// TIA Portal V16 export
// export: Created 2022-04-06T03:32:48.1224576Z, ExportSetting WithDefaults, DisplayName Totally Integrated Automation Portal, DisplayVersion V16 Update 4, DisplayName TIA Portal Version Control Interface, DisplayVersion V16 Update 2, DisplayName TIA Portal Openness, DisplayVersion V16 Update 4, DisplayName SINAMICS Startdrive Advanced, DisplayVersion V16, DisplayName SINAMICS Startdrive G130, G150, S120, S150, SINAMICS MV, S210, DisplayVersion V16, DisplayName SINAMICS Startdrive G110M, G120, G120C, G120D, G120P, DisplayVersion V16, DisplayName STEP 7 Professional, DisplayVersion V16 Update 4, DisplayName STEP 7 Safety, DisplayVersion V16, DisplayName WinCC Professional, DisplayVersion V16 Update 4
FUNCTION_BLOCK "fbRoomHVAC"   // FB7, LAD
{ S7_Optimized_Access := 'TRUE' }
VERSION : 0.1
// stored: AutoNumber true, IsIECCheckEnabled false, IsRetainMemResEnabled false, MemoryReserve 100, SetENOAutomatically false, UDAEnableTagReadback false
   VAR
      Temperature_Cooling { ExternalVisible := 'False'} : "fbAlarmedSetpoint";
      Humidity { ExternalVisible := 'False'} : "fbAlarmedSetpoint";
      CO2 { S7_SetPoint := 'True'} : "fbAlarmedSetpoint";
   END_VAR
   VAR RETAIN
      Controls { ExternalVisible := 'False'} : Struct
         rHeatingSP { ExternalVisible := 'False'} : Real := 55.0;
         bResetAlarm { ExternalVisible := 'False'} : Bool;
         bResetModbus { ExternalVisible := 'False'} : Bool;
      END_STRUCT;
      Status { ExternalVisible := 'False'; ExternalWritable := 'False'} : Struct
         bModbusError { ExternalVisible := 'False'; ExternalWritable := 'False'} : Bool;
         wLastModbusErrorCode { ExternalVisible := 'False'; ExternalWritable := 'False'} : Word;
      END_STRUCT;
      Config { ExternalVisible := 'False'} : Struct
         ModbusServerAddr { ExternalVisible := 'False'} : IP_V4;   // IP address for Modbus TCP server
         ID { ExternalVisible := 'False'} : UInt := 81;   // Unique ID for connection, also used as port number on PLC
      END_STRUCT;
   END_VAR
   VAR
      TCPConnection { ExternalAccessible := 'False'; ExternalVisible := 'False'; ExternalWritable := 'False'} : TCON_IP_v4;
      fbModbusTCPClient_Instance { ExternalAccessible := 'False'; ExternalVisible := 'False'; ExternalWritable := 'False'} : "fbModbusTCPClient";
      Read_Discrete { ExternalAccessible := 'False'; ExternalVisible := 'False'; ExternalWritable := 'False'} : Array[0..0] of "udtModbusValBool";
      Write_Discrete { ExternalAccessible := 'False'; ExternalVisible := 'False'; ExternalWritable := 'False'} : Array[0..0] of "udtModbusValBool";
      Read_Registers { ExternalAccessible := 'False'; ExternalVisible := 'False'; ExternalWritable := 'False'} : Array[0..2] of "udtModbusValReal";
      Write_Registers { ExternalAccessible := 'False'; ExternalVisible := 'False'; ExternalWritable := 'False'} : Array[0..2] of "udtModbusValReal";
      TON_ModbusReset { S7_SetPoint := 'True'} : TON_TIME;
      mbreset { ExternalAccessible := 'False'; ExternalVisible := 'False'; ExternalWritable := 'False'} : Bool;
      TP_ModbusResetPulse { S7_SetPoint := 'True'} : TP_TIME;
   END_VAR
   VAR CONSTANT
      cFakeScaling : Int := 150;
      cRoomTempIndex : Int := 0;
      cHumidityIndex : Int := 1;
      cCO2Index : Int := 2;
   END_VAR
   // Temperature_Cooling.arrSetpoints[1].rSetpoint := 75.0;
   // Humidity.arrSetpoints[1].rSetpoint := 55.0;
   // Config.ModbusServerAddr.ADDR[1] := 10;
   // Config.ModbusServerAddr.ADDR[2] := 1;
   // Config.ModbusServerAddr.ADDR[3] := 0;
   // Config.ModbusServerAddr.ADDR[4] := 8;
   // TCPConnection.ConnectionType := 11;
   // TCPConnection.ActiveEstablished := true;
   // TCPConnection.RemoteAddress.ADDR[1] := 10;
   // TCPConnection.RemoteAddress.ADDR[2] := 1;
   // TCPConnection.RemoteAddress.ADDR[3] := 2;
   // TCPConnection.RemoteAddress.ADDR[4] := 8;
   // TCPConnection.RemotePort := 502;
   // TCPConnection.LocalPort := 1001;
BEGIN

REGION Network 1 (SCL): Set connection parameters
   #TCPConnection.InterfaceId := "Local~PROFINET_interface_1"; // PLC ethernet port
   #TCPConnection.ID := UINT_TO_WORD(#Config.ID);
   #TCPConnection.ConnectionType := 11; // TCP
   #TCPConnection.ActiveEstablished := TRUE;
   #TCPConnection.RemoteAddress := #Config.ModbusServerAddr;
   #TCPConnection.RemotePort := 502; // Default for Modbus TCP
   #TCPConnection.LocalPort := #Config.ID;
END_REGION

REGION Network 2 (SCL): Reset Modbus on Error

   #mbreset := #TON_ModbusReset.Q;
   #TON_ModbusReset(IN := #Status.bModbusError AND NOT #mbreset,
                    PT := T#10S);

   #TP_ModbusResetPulse(IN:=#mbreset,
                        PT:=T#5S,
                        Q => #Controls.bResetModbus);
END_REGION

REGION Network 3 (SCL): Set up registers
   // Read coils and discrete inputs (00001 and 10001)
   //#Read_Discrete[0].iAddr := 00045;

   // Write coils (00001)
   //#Write_Discrete[0].iAddr := 00191; 
   //#Write_Discrete[0].bVal := 0;

   // Read input and holding registers (30001 and 40001)
   #Read_Registers[cRoomTempIndex].iRegister := 30002; // Room Temperature // should be 30001
   #Read_Registers[cHumidityIndex].iRegister := 35004; // Humidity
   #Read_Registers[cCO2Index].iRegister := 35182;  // CO2

   // Write holding registers (40001)
   #Write_Registers[0].iRegister := 40005; // Cooling SP
   #Write_Registers[0].rVal := #Temperature_Cooling.rSetpoint * 10; // re-scale due to gPod bs

   #Write_Registers[1].iRegister := 45185; // CO2 SP
   #Write_Registers[1].rVal := #CO2.rSetpoint;

   #Write_Registers[2].iRegister := 45030; // Dehumidification SP
   #Write_Registers[2].rVal := #Humidity.rSetpoint;
END_REGION

REGION Network 4: Modbus TCP Client Block Call
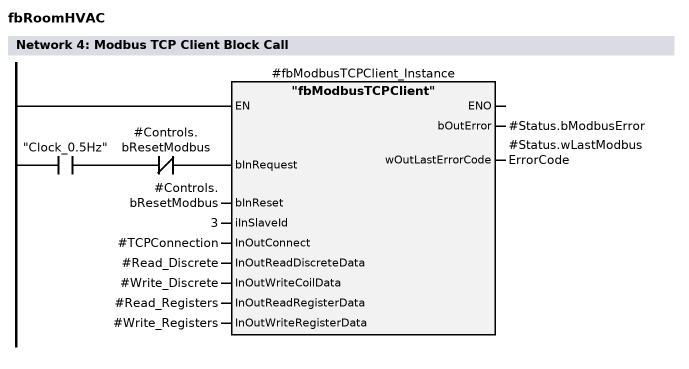
   RUNG wire#powerrail
      #fbModbusTCPClient_Instance(bInRequest := wire#w1, bInReset := #Controls.bResetModbus, iInSlaveId := 3, InOutConnect := #TCPConnection, InOutReadDiscreteData := #Read_Discrete, InOutWriteCoilData := #Write_Discrete, InOutReadRegisterData := #Read_Registers, InOutWriteRegisterData := #Write_Registers, bOutError => #Status.bModbusError, wOutLastErrorCode => #Status.wLastModbusErrorCode)
   END_RUNG
   RUNG wire#powerrail
      Contact( "Clock_0.5Hz" )
      I_Contact( #Controls.bResetModbus )
   END_RUNG wire#w1
   // the same network as SCL:
   #fbModbusTCPClient_Instance(bInRequest := "Clock_0.5Hz" AND NOT #Controls.bResetModbus,   // "fbModbusTCPClient"
                           bInReset := #Controls.bResetModbus,
                           iInSlaveId := 3,
                           InOutConnect := #TCPConnection,
                           InOutReadDiscreteData := #Read_Discrete,
                           InOutWriteCoilData := #Write_Discrete,
                           InOutReadRegisterData := #Read_Registers,
                           InOutWriteRegisterData := #Write_Registers,
                           bOutError => #Status.bModbusError,
                           wOutLastErrorCode => #Status.wLastModbusErrorCode);
END_REGION

REGION Network 5 (SCL): Parse received data


   #Temperature_Cooling(iInRawValue := #Read_Registers[cRoomTempIndex].rVal * 0.1); // the value from the gPod requires scaling in this way
   #Humidity(iInRawValue := #Read_Registers[cHumidityIndex].rVal);
   #CO2(iInRawValue := #Read_Registers[cCO2Index].rVal);
END_REGION
END_FUNCTION_BLOCK
